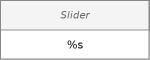
VISUALIZATION UC_Slider  // 150x60
VAR_IN_OUT
	PT		:TIME;
END_VAR
VAR_INPUT
	Start,End,MainScale	:UDINT;
	Label				:STRING;
END_VAR
    Slider (0,0 150x30), variable: PT, scale 0..1000
    Textfield (0,30 150x30), "%s", text variable: Label
END_VISUALIZATION

(* stored: Version 1.1.0.1
   Visu UC_Slider: Id {eda1783a-037a-44ee-89b4-e851fcff7e76} *)
